// TwinCAT 3 PLC project ServerSampleProject
// ProgramVersion: 3.1.0.8
// libraries:
//   Tc2_Standard, * (Beckhoff Automation GmbH)
//   Tc2_System, * (Beckhoff Automation GmbH)
//   Tc3_Interfaces, * (Beckhoff Automation GmbH)
//   Tc3_Module, * (Beckhoff Automation GmbH)
// project tree:
//   DUTs/ ST_Structure.TcDUT, ST_SubStructure.TcDUT
//   / PlcTask.TcTTO (not stored)
//   POUs/ FB_Mathematics.TcPOU (not stored), MAIN.TcPOU
// real-time tasks:
//   TASK PlcTask: cycle T#10ms, priority 20, ADS port 350

// ---- DUTs/ST_Structure.TcDUT
TYPE ST_Structure :
STRUCT
	a : INT;
	b : DINT;
	c : ARRAY[0..9] OF REAL;
	{attribute 'OPC.UA.DA.StructuredType':='1'}
	d : ST_SubStructure;
END_STRUCT
END_TYPE

// ---- DUTs/ST_SubStructure.TcDUT
TYPE ST_SubStructure :
STRUCT
	e : LREAL;
	f : DT;
END_STRUCT
END_TYPE

// ---- POUs/MAIN.TcPOU
PROGRAM MAIN
VAR
	{attribute 'OPC.UA.DA':='1'}
	nCounter : INT;
	
	{attribute 'OPC.UA.DA':='1'}
	nNumber : INT;
	
	{attribute 'OPC.UA.DA':='1'}
	fbMathematics : FB_Mathematics;
	
	{attribute 'OPC.UA.DA':='1'}
	iVar1 : INT := 42;
	
	{attribute 'OPC.UA.DA':='1'}
	iVar2 : INT := 43;
	
	{attribute 'OPC.UA.DA':='1'}
	{attribute 'OPC.UA.DA.Access':='1'}
	iVar3_readOnly : INT := 43;	
	
	{attribute 'OPC.UA.DA':='1'}
	{attribute 'OPC.UA.DA.Description' := 'Some description'} 
	iArrayIntVar1 : ARRAY[0..9] OF INT := [10(42)];
	
	{attribute 'OPC.UA.DA':='1'}
	iArrayIntVar2 : ARRAY[0..11] OF INT := [12(41)];	
	
	{attribute 'OPC.UA.DA':='1'}
	iArrayIntVar3 : ARRAY[0..9] OF DINT;
	
	{attribute 'OPC.UA.DA':='1'}
	{attribute 'OPC.UA.DA.StructuredType':='1'}
	stStructure : ST_Structure;
END_VAR

nCounter := nCounter + 1;

END_PROGRAM
